(* PLC project Tc2_Utilities.FB_GetLicenseDongles Demo, tc3-libraries-kb TwinCAT 3.1 *)
(* stored: creationDateTime 2026-05-11T00:00:00, modificationDateTime 2026-05-11T00:00:00 *)

PROGRAM P_Demo_FB_GetLicenseDongles
  VAR
    fbFB_GetLicenseDongles : FB_GetLicenseDongles;  (* FB_GetLicenseDongles 实例 *)
    bExec : BOOL := FALSE;
    bBusy_ : BOOL;
    bErrFlag : BOOL;
    nErrCode : UDINT;
  END_VAR

// =============================================================================
// 场景：多 dongle 列出。
// 价值：多 dongle 环境管理。
// 验证：触发后观察 bDone / bErr，错误号 nErrId 反映 ADS Return Codes。
// 验证步骤：
//   1. 右键 PLC 项目 → Import PLCopenXML → 选本文件
//   2. 引用 Tc2_Utilities（References → Add library）
//   3. 编译 → 登录 → 运行；按上方『验证』行的指示在线写值观察
// =============================================================================

fbFB_GetLicenseDongles(
    bExecute := bExec, tTimeout := DEFAULT_ADS_TIMEOUT,
    bBusy => bBusy_, bError => bErrFlag, nErrorId => nErrCode
);
END_PROGRAM
